// TIA Portal V18 export
FUNCTION "Metering Program sequences" : Void   // FC2, LAD
{ S7_Optimized_Access := 'TRUE' }
VERSION : 0.1
// stored: AutoNumber true, IsIECCheckEnabled false, SetENOAutomatically false, UDAEnableTagReadback false
   VAR_TEMP
      temp1 : Bool;
   END_VAR
   VAR_TEMP   // added for the SCL form of the ladder/FBD networks
      _w1 : Bool;
   END_VAR
BEGIN

REGION Network 1: Do continous metering selection
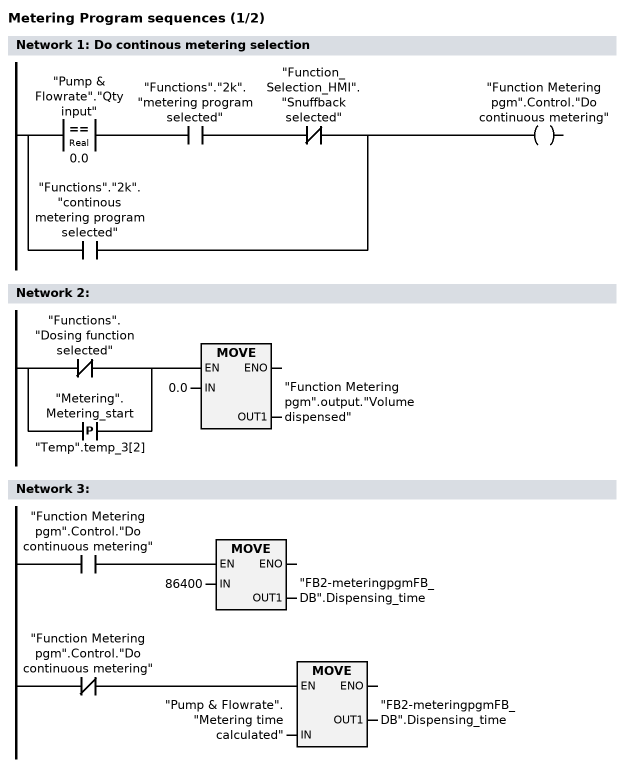
   RUNG wire#powerrail
      { S7_Templates := "SrcType := Real" } EQ_Contact(in1 := "Pump & Flowrate"."Qty input", in2 := 0.0)
      Contact( "Functions"."2k"."metering program selected" )
      I_Contact( "Function_Selection_HMI"."Snuffback selected" )
      wire#w1
      Coil( "Function Metering pgm".Control."Do continuous metering" )
   END_RUNG
   RUNG wire#powerrail
      Contact( "Functions"."2k"."continous metering program selected" )
   END_RUNG wire#w1
   // the same network as SCL:
   "Function Metering pgm".Control."Do continuous metering" := (("Pump & Flowrate"."Qty input" = 0.0) AND "Functions"."2k"."metering program selected" AND NOT "Function_Selection_HMI"."Snuffback selected") OR "Functions"."2k"."continous metering program selected";
END_REGION

REGION Network 2
   RUNG wire#powerrail
      I_Contact( "Functions"."Dosing function selected" )
      wire#w1
      Move(in := 0.0, out1 => "Function Metering pgm".output."Volume dispensed")
   END_RUNG
   RUNG wire#powerrail
      P_Contact(operand := "Metering".Metering_start, bit := "Temp".temp_3[2])
   END_RUNG wire#w1
   // the same network as SCL:
   #_w1 := "Metering".Metering_start AND NOT "Temp".temp_3[2];   // rising edge of "Metering".Metering_start
   "Temp".temp_3[2] := "Metering".Metering_start;
   IF NOT "Functions"."Dosing function selected" OR #_w1 THEN
       "Function Metering pgm".output."Volume dispensed" := 0.0;
   END_IF;
END_REGION

REGION Network 3
   RUNG wire#powerrail
      Contact( "Function Metering pgm".Control."Do continuous metering" )
      Move(in := 86400, out1 => "FB2-meteringpgmFB_DB".Dispensing_time)
   END_RUNG
   RUNG wire#powerrail
      I_Contact( "Function Metering pgm".Control."Do continuous metering" )
      Move(in := "Pump & Flowrate"."Metering time calculated", out1 => "FB2-meteringpgmFB_DB".Dispensing_time)
   END_RUNG
   // the same network as SCL:
   IF "Function Metering pgm".Control."Do continuous metering" THEN
       "FB2-meteringpgmFB_DB".Dispensing_time := 86400;
   END_IF;
   IF NOT "Function Metering pgm".Control."Do continuous metering" THEN
       "FB2-meteringpgmFB_DB".Dispensing_time := "Pump & Flowrate"."Metering time calculated";
   END_IF;
END_REGION

REGION Network 4
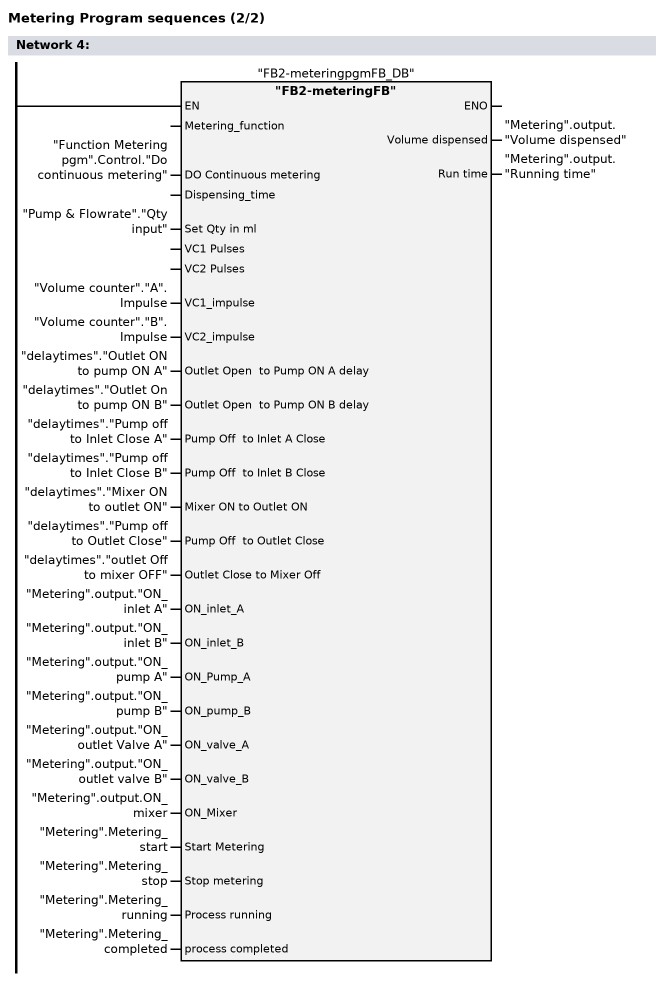
   RUNG wire#powerrail
      "FB2-meteringpgmFB_DB"(Metering_function :=, "DO Continuous metering" := "Function Metering pgm".Control."Do continuous metering", Dispensing_time :=, "Set Qty in ml" := "Pump & Flowrate"."Qty input", "VC1 Pulses" :=, "VC2 Pulses" :=, VC1_impulse := "Volume counter"."A".Impulse, VC2_impulse := "Volume counter"."B".Impulse, "Outlet Open  to Pump ON A delay" := "delaytimes"."Outlet ON to pump ON A", "Outlet Open  to Pump ON B delay" := "delaytimes"."Outlet On to pump ON B", "Pump Off  to Inlet A Close" := "delaytimes"."Pump off to Inlet Close A", "Pump Off  to Inlet B Close" := "delaytimes"."Pump off to Inlet Close B", "Mixer ON to Outlet ON" := "delaytimes"."Mixer ON to outlet ON", "Pump Off  to Outlet Close" := "delaytimes"."Pump off to Outlet Close", "Outlet Close to Mixer Off" := "delaytimes"."outlet Off to mixer OFF", ON_inlet_A := "Metering".output."ON_inlet A", ON_inlet_B := "Metering".output."ON_inlet B", ON_Pump_A := "Metering".output."ON_pump A", ON_pump_B := "Metering".output."ON_pump B", ON_valve_A := "Metering".output."ON_outlet Valve A", ON_valve_B := "Metering".output."ON_outlet valve B", ON_Mixer := "Metering".output.ON_mixer, "Start Metering" := "Metering".Metering_start, "Stop metering" := "Metering".Metering_stop, "Process running" := "Metering".Metering_running, "process completed" := "Metering".Metering_completed, "Volume dispensed" => "Metering".output."Volume dispensed", "Run time" => "Metering".output."Running time")
   END_RUNG
   // the same network as SCL:
   "FB2-meteringpgmFB_DB"("DO Continuous metering" := "Function Metering pgm".Control."Do continuous metering",   // "FB2-meteringFB"
                          "Set Qty in ml" := "Pump & Flowrate"."Qty input",
                          VC1_impulse := "Volume counter"."A".Impulse,
                          VC2_impulse := "Volume counter"."B".Impulse,
                          "Outlet Open  to Pump ON A delay" := "delaytimes"."Outlet ON to pump ON A",
                          "Outlet Open  to Pump ON B delay" := "delaytimes"."Outlet On to pump ON B",
                          "Pump Off  to Inlet A Close" := "delaytimes"."Pump off to Inlet Close A",
                          "Pump Off  to Inlet B Close" := "delaytimes"."Pump off to Inlet Close B",
                          "Mixer ON to Outlet ON" := "delaytimes"."Mixer ON to outlet ON",
                          "Pump Off  to Outlet Close" := "delaytimes"."Pump off to Outlet Close",
                          "Outlet Close to Mixer Off" := "delaytimes"."outlet Off to mixer OFF",
                          ON_inlet_A := "Metering".output."ON_inlet A",
                          ON_inlet_B := "Metering".output."ON_inlet B",
                          ON_Pump_A := "Metering".output."ON_pump A",
                          ON_pump_B := "Metering".output."ON_pump B",
                          ON_valve_A := "Metering".output."ON_outlet Valve A",
                          ON_valve_B := "Metering".output."ON_outlet valve B",
                          ON_Mixer := "Metering".output.ON_mixer,
                          "Start Metering" := "Metering".Metering_start,
                          "Stop metering" := "Metering".Metering_stop,
                          "Process running" := "Metering".Metering_running,
                          "process completed" := "Metering".Metering_completed,
                          "Volume dispensed" => "Metering".output."Volume dispensed",
                          "Run time" => "Metering".output."Running time");
END_REGION

REGION Network 5 (SCL)
   //IF NOT ("Gear Pump B On_REW") AND NOT ("Gear Pump A On_REW") THEN
       IF "Functions"."2k"."continous metering program selected" THEN
           "Function Continous Metering pgm".output."Volume dispensed" := "Metering".output."Volume dispensed";
           "Function Continous Metering pgm".output."Running time" := "Metering".output."Running time";
       ELSIF "Functions"."2k"."metering program selected" THEN
           "Function Metering pgm".output."Volume dispensed" := "Metering".output."Volume dispensed";
           "Function Metering pgm".output."Running time" := "Metering".output."Running time";
       ELSIF "Functions"."2k"."shot metering program selected" THEN
           "Function shot Metering".output."Volume dispensed" := "Metering".output."Volume dispensed";
           "Function shot Metering".output."Running time" := "Metering".output."Running time";
       ELSIF "Functions"."2k"."pre run program selected" THEN
           "Function Pre run".output."Volume dispensed" := "Metering".output."Volume dispensed";
           "Function Pre run".output."Running time" := "Metering".output."Running time";
       END_IF;
   //END_IF;
END_REGION

REGION Network 6 (SCL): Prerun Completed
   IF "Functions"."2k"."pre run program selected" AND "Metering".Metering_completed THEN //AND  ("Function Pre run".output."Volume dispensed" >="Pump & Flowrate"."Qty input")
       "Function Pre run".Control."metering completed" := TRUE;
   ELSIF "Function Flush"."Control A"."flush running" OR "Function Dearing with valve"."Control A"."dearing running"
       OR "Function Dearing with valve"."Control B"."dearing running" OR "Potlife".contol."Potlife elapsed machine not in regeneration"
           THEN //OR ("Functions"."2k"."pre run program selected"  AND "Functions"."Stop Dosing function")

       "Function Pre run".Control."metering completed" := FALSE;
   END_IF;
   "Control"."waiting For pre run" := NOT ("Function Pre run".Control."metering completed");
END_REGION
END_FUNCTION
